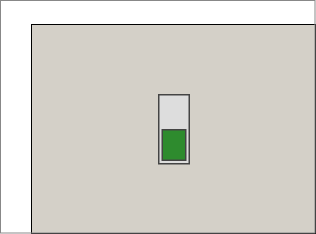
VISUALIZATION Visualization  // 316x234
    Rectangle (31,24 285x210)
    DipSwitch (139,94 70x70), variable: MAIN.bRun, behaviour: TOGGLE, style: Switch-DipSwitch-Green
END_VISUALIZATION

(* stored: Version 1.1.0.1, ProductVersion 3.1.4024.13
   Visu Visualization: Id {ca9fa920-428c-4b46-b467-f65363b83988} *)
